Universal Robots PolyScope program: Program1.urp

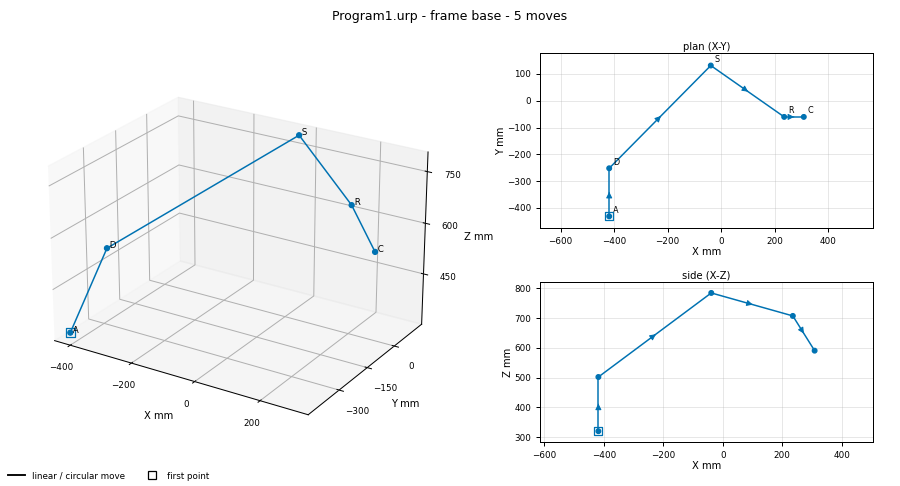
[picture p0: tool path of Program1.urp in frame base, 5 of 5 moves have a stored position in this frame; points joined in program order, loops and branches not executed]
Program Program1 (installation=default directory=/ursim/programs createdIn=3.15.8.106339 lastSavedIn=3.15.8.106339 robotSerialNumber=2018359999)
Calibrated DH parameters: a=[0, -0.425, -0.39225, 0, 0, 0]; d=[0.089159, 0, 0, 0.10915, 0.09465, 0.0823]; alpha=[1.570796, 0, 0, 1.570796, -1.570796, 0]; deltaTheta=[0, 0, 0, 0, 0, 0]
InitVariablesNode
Robot Program (runOnlyOnce=false)
  Popup Message (haltProgram=false message=Iniciamos con el programa 1, INICIALES INTEGRANTES inputType=Text)
  MoveL speed 250 mm/s, acceleration 1200 mm/s^2 (useActiveTCP=true) feature=Base
    Waypoint A: TCP in base x=-418.111 y=-431.763 z=319.671 mm, rx=-0.0012 ry=3.1163 rz=0.0389 rad; joints [-123.672, -106.14, -87.456, -78.391, 90.402, -33.724] deg
    Popup Message (haltProgram=false message=Finalizacion letra A e inicio letra S inputType=Text)
    MoveL speed 250 mm/s, acceleration 1200 mm/s^2 (useActiveTCP=true) feature=Base
      Waypoint D: TCP in base x=-418.111 y=-252.165 z=501.832 mm, rx=-0.007 ry=-2.6954 rz=-0.0338 rad; joints [-132.654, -85.282, -89.475, -78.353, 70.484, -45.282] deg
      Popup Message (haltProgram=false message=Finalizacion D e inicio S inputType=Text)
      MoveL speed 250 mm/s, acceleration 1200 mm/s^2 (useActiveTCP=true) feature=Base
        Waypoint S: TCP in base x=-38.675 y=131.615 z=784.4 mm, rx=-1.1756 ry=-1.3707 rz=0.6075 rad; joints [-180.637, -46.156, -81.175, -64.239, 74.476, -22.093] deg
        Popup Message (haltProgram=false message=Finalizacion de S e inicio de R inputType=Text)
        MoveL speed 250 mm/s, acceleration 1200 mm/s^2 (useActiveTCP=true) feature=Base
          Waypoint R: TCP in base x=235.477 y=-60.286 z=707.187 mm, rx=-1.3 ry=-0.4525 rz=0.0727 rad; joints [-228.523, -19.791, -91.465, -56.907, 70.594, -20.688] deg
          Popup Message (haltProgram=false message=Finalizacion de R e inicio de C inputType=Text)
          MoveL speed 250 mm/s, acceleration 1200 mm/s^2 (useActiveTCP=true) feature=Base
            Waypoint C: TCP in base x=308.731 y=-60.286 z=590.387 mm, rx=-1.3 ry=-0.4525 rz=0.0727 rad; joints [-219.205, -1.767, -102.664, -62.85, 61.489, -22.854] deg
  Popup Message (haltProgram=false message=Terminamos programa 1 e iniciamos programa 2 inputType=Text)
